FUNCTION_BLOCK PUBLIC StackForwardEnumerator_TestSuite EXTENDS TcUnit.FB_TestSuite

CheckIsValidAtStart();
CheckMoveNextReturnsFalseAtTheEnd();
CheckMoveNextReturnsFalseWhenEmpty();
CheckMoveNextReturnsTrueMultipleItems();
CheckMoveNextReturnsTrueSingleItem();
CheckReset();
CheckTryGet();
CheckTryGetTo();
CheckWorksWithIntegers();
CheckWorksWithStrings();
CheckWorksWithArrays();

METHOD PUBLIC CheckIsValidAtStart
VAR
	result : BOOL;
	stack : Stack;
	enumerator : I_ForwardEnumerator;
END_VAR
TEST('CheckIsValidAtStart');

enumerator := stack.GetEnumerator();

result := enumerator.IsValid;
enumerator.Dispose();

AssertTrue(
	Condition := result,
	Message := 'Method returned false'
);

TEST_FINISHED();
END_METHOD

METHOD PRIVATE CheckMoveNextReturnsFalseAtTheEnd
VAR
	in1 : INT := 123;
	result : BOOL;
	stack : Stack;
	enumerator : I_ForwardEnumerator;
END_VAR
TEST('CheckMoveNextReturnsFalseAtTheEnd');

stack.Push(in1);
enumerator := stack.GetEnumerator();

enumerator.MoveNext();
result := enumerator.MoveNext();
enumerator.Dispose();

AssertFalse(result,
    'MoveNext did not correctly signal the end of the enumeration');
	
TEST_FINISHED();
END_METHOD

METHOD PUBLIC CheckMoveNextReturnsFalseWhenEmpty
VAR
	result : BOOL;
	stack : Stack;
	enumerator : I_ForwardEnumerator;
END_VAR
TEST('CheckMoveNextReturnsFalseWhenEmpty');

enumerator := stack.GetEnumerator();

result := enumerator.MoveNext();
enumerator.Dispose();

AssertFalse(
	Condition := result,
	Message := 'MoveNext did not correctly signal the end of the enumeration'
);

TEST_FINISHED();
END_METHOD

METHOD PRIVATE CheckMoveNextReturnsTrueMultipleItems
VAR
	in1 : INT := 123;
	in2 : INT := 456;
	in3 : INT := 789;
	result : BOOL;
	stack : Stack;
	enumerator : I_ForwardEnumerator;
END_VAR
TEST('CheckMoveNextReturnsTrueMultipleItems');

stack.Push(in1);
stack.Push(in2);
stack.Push(in3);
enumerator := stack.GetEnumerator();

result := enumerator.MoveNext();
enumerator.Dispose();

AssertTrue(result, 'MoveNext did not correctly signal there were more items to follow');

TEST_FINISHED();
END_METHOD

METHOD PRIVATE CheckMoveNextReturnsTrueSingleItem
VAR
	in1 : INT := 123;
	result : BOOL;
	stack : Stack;
	enumerator : I_ForwardEnumerator;
END_VAR
TEST('CheckMoveNextReturnsTrueSingleItem');

stack.Push(in1);
enumerator := stack.GetEnumerator();

result := enumerator.MoveNext();
enumerator.Dispose();

AssertTrue(result,
    'MoveNext did not correctly signal there were more items to follow');
	
TEST_FINISHED();
END_METHOD

METHOD PUBLIC CheckReset
VAR
	in1 : ARRAY [0..1] OF REAL := [0.1,2.3];
	in2 : ARRAY [0..1] OF REAL := [1.2,3.4];
	in3 : ARRAY [0..1] OF REAL := [2.3,4.5];
	out : ARRAY [0..1] OF REAL;
	expected : ARRAY [0..1] OF REAL := [2.3,4.5];
	stack : Stack;
	enumerator : I_ForwardEnumerator;
END_VAR
TEST('CheckReset');

stack.Push(in1);
stack.Push(in2);
stack.Push(in3);

enumerator := stack.GetEnumerator();

enumerator.MoveNext();
enumerator.MoveNext();
enumerator.Reset();
enumerator.MoveNext();
enumerator.TryGet(out);

enumerator.Dispose();

AssertEquals(
	Expected := expected,
	Actual := out,
	Message := 'Did not produce the expected result'
);

TEST_FINISHED();
END_METHOD

METHOD PUBLIC CheckTryGet
VAR
	in : INT := 123;
	out : INT;
	expected : INT := 123;
	result : BOOL;
	stack : Stack;
	enumerator : I_ForwardEnumerator;
END_VAR
TEST('CheckTryGet');

stack.Push(in);
enumerator := stack.GetEnumerator();
enumerator.MoveNext();

result := enumerator.TryGet(out);
enumerator.Dispose();

AssertTrue(
	Condition := result,
	Message := 'Method returned false'
);

AssertEquals(
	Expected := expected,
	Actual := out,
	Message := 'Did not produce the expected result'
);

TEST_FINISHED();
END_METHOD

METHOD PUBLIC CheckTryGetTo
VAR
	in : INT := 123;
	out : INT;
	expected : INT := 123;
	result : BOOL;
	stack : Stack;
	enumerator : I_ForwardEnumerator;
END_VAR
TEST('CheckTryGetTo');

stack.Push(in);
enumerator := stack.GetEnumerator();
enumerator.MoveNext();

result := enumerator.TryGetTo(ADR(out),SIZEOF(out));
enumerator.Dispose();

AssertTrue(
	Condition := result,
	Message := 'Method returned false'
);

AssertEquals(
	Expected := expected,
	Actual := out,
	Message := 'Did not produce the expected result'
);

TEST_FINISHED();
END_METHOD

METHOD PUBLIC CheckWorksWithArrays
VAR
	in1 : ARRAY [0..1] OF REAL := [0.1,2.3];
	in2 : ARRAY [0..1] OF REAL := [1.2,3.4];
	in3 : ARRAY [0..1] OF REAL := [2.3,4.5];
	out1 : ARRAY [0..1] OF REAL;
	out2 : ARRAY [0..1] OF REAL;
	out3 : ARRAY [0..1] OF REAL;
	expected1 : ARRAY [0..1] OF REAL := [2.3,4.5];
	expected2 : ARRAY [0..1] OF REAL := [1.2,3.4];
	expected3 : ARRAY [0..1] OF REAL := [0.1,2.3];
	stack : Stack;
	enumerator : I_ForwardEnumerator;
END_VAR
TEST('CheckWorksWithArrays');

stack.Push(in1);
stack.Push(in2);
stack.Push(in3);

enumerator := stack.GetEnumerator();

enumerator.MoveNext();
enumerator.TryGet(out1);
enumerator.MoveNext();
enumerator.TryGet(out2);
enumerator.MoveNext();
enumerator.TryGet(out3);

enumerator.Dispose();

AssertEquals(
	Expected := expected1,
	Actual := out1,
	Message := 'Did not produce the expected 1st result'
);

AssertEquals(
	Expected := expected2,
	Actual := out2,
	Message := 'Did not produce the expected 2nd result'
);

AssertEquals(
	Expected := expected3,
	Actual := out3,
	Message := 'Did not produce the expected 3rd result'
);

TEST_FINISHED();
END_METHOD

METHOD PUBLIC CheckWorksWithIntegers
VAR
	in1 : INT := 123;
	in2 : INT := 234;
	in3 : INT := 345;
	out1 : INT;
	out2 : INT;
	out3 : INT;
	expected1 : INT := 345;
	expected2 : INT := 234;
	expected3 : INT := 123;
	stack : Stack;
	enumerator : I_ForwardEnumerator;
END_VAR
TEST('CheckWorksWithIntegers');

stack.Push(in1);
stack.Push(in2);
stack.Push(in3);

enumerator := stack.GetEnumerator();

enumerator.MoveNext();
enumerator.TryGet(out1);
enumerator.MoveNext();
enumerator.TryGet(out2);
enumerator.MoveNext();
enumerator.TryGet(out3);

enumerator.Dispose();

AssertEquals(
	Expected := expected1,
	Actual := out1,
	Message := 'Did not produce the expected 1st result'
);

AssertEquals(
	Expected := expected2,
	Actual := out2,
	Message := 'Did not produce the expected 2nd result'
);

AssertEquals(
	Expected := expected3,
	Actual := out3,
	Message := 'Did not produce the expected 3rd result'
);

TEST_FINISHED();
END_METHOD

METHOD PUBLIC CheckWorksWithStrings
VAR
	in1 : STRING := 'test1';
	in2 : STRING := 'test2';
	in3 : STRING := 'test3';
	out1 : STRING;
	out2 : STRING;
	out3 : STRING;
	expected1 : STRING := 'test3';
	expected2 : STRING := 'test2';
	expected3 : STRING := 'test1';
	stack : Stack;
	enumerator : I_ForwardEnumerator;
END_VAR
TEST('CheckWorksWithStrings');

stack.Push(in1);
stack.Push(in2);
stack.Push(in3);

enumerator := stack.GetEnumerator();

enumerator.MoveNext();
enumerator.TryGet(out1);
enumerator.MoveNext();
enumerator.TryGet(out2);
enumerator.MoveNext();
enumerator.TryGet(out3);

enumerator.Dispose();

AssertEquals(
	Expected := expected1,
	Actual := out1,
	Message := 'Did not produce the expected 1st result'
);

AssertEquals(
	Expected := expected2,
	Actual := out2,
	Message := 'Did not produce the expected 2nd result'
);

AssertEquals(
	Expected := expected3,
	Actual := out3,
	Message := 'Did not produce the expected 3rd result'
);

TEST_FINISHED();
END_METHOD

END_FUNCTION_BLOCK

(* stored: Version 1.1.0.1, ProductVersion 3.1.4024.12
   POU StackForwardEnumerator_TestSuite: Id {307ab2e6-2fb6-45e5-81fd-4e16fa1b1495}, SpecialFunc None
   Method CheckIsValidAtStart: Id {3c7b1a75-4448-407f-b8e5-7af5a5403c62}
   Method CheckMoveNextReturnsFalseAtTheEnd: Id {e9d8cbda-4018-40d6-96f3-95f470d3a50a}
   Method CheckMoveNextReturnsFalseWhenEmpty: Id {88e27552-8a43-400f-8ffa-e2fef0fa0b48}
   Method CheckMoveNextReturnsTrueMultipleItems: Id {77378285-00e5-40b0-b0b4-9331da50f447}
   Method CheckMoveNextReturnsTrueSingleItem: Id {0191ceb7-6602-4ffc-8e87-0603a5ec0915}
   Method CheckReset: Id {c1938e5f-dbd2-4e10-aad4-c673be0da618}
   Method CheckTryGet: Id {286c6be9-05b0-4d83-a7fb-546bec4a8d3b}
   Method CheckTryGetTo: Id {dd708e17-5aeb-453e-bc47-465f1175c4fb}
   Method CheckWorksWithArrays: Id {8dbbc900-5cbd-4129-afee-f06f6abd7f4c}
   Method CheckWorksWithIntegers: Id {4abcc6e8-e3e6-4604-8b5f-90e6f8bbba44}
   Method CheckWorksWithStrings: Id {5b4ac783-359e-4250-a936-191ee4c0ecfc} *)
